PROGRAM P_RunClock
VAR
	fbRunClock : FB_RunClock;
END_VAR

fbRunClock(
	bStart := TRUE,
	bStop := G_Inputs.bStopButton,
	fCycleTime := G_Parameter.fCycleTime,
	
	fTime => G_OPC.fTime
);

END_PROGRAM

(* stored: Version 1.1.0.1, ProductVersion 3.1.4024.12
   POU P_RunClock: Id {d8c930b5-bf90-4658-99e0-6b7148646632}, SpecialFunc None *)
